//     Term 17 (AT2000-0250)/Term 18 (AT2000-5250)/FB Inputs/Value Channel 26 <-> Data Pointer/RawPositionValues[25]
//     Term 17 (AT2000-0250)/Term 18 (AT2000-5250)/FB Inputs/Value Channel 27 <-> Data Pointer/RawPositionValues[26]
//     Term 17 (AT2000-0250)/Term 18 (AT2000-5250)/FB Inputs/Value Channel 28 <-> Data Pointer/RawPositionValues[27]
//     Term 17 (AT2000-0250)/Term 18 (AT2000-5250)/FB Inputs/Value Channel 29 <-> Data Pointer/RawPositionValues[28]
//     Term 17 (AT2000-0250)/Term 18 (AT2000-5250)/FB Inputs/Value Channel 30 <-> Data Pointer/RawPositionValues[29]
//     Term 17 (AT2000-0250)/Term 18 (AT2000-5250)/FB Inputs/Value Channel 31 <-> Data Pointer/RawPositionValues[30]
//     Term 17 (AT2000-0250)/Term 18 (AT2000-5250)/FB Inputs/Value Channel 32 <-> Data Pointer/RawPositionValues[31]
//   NC-Task 1 SAF/Axes/Mover Axis 1 <-> TcCOM Objects/XTS ProcessingUnit 1/Mover 1
//     SoftDrive 1/Data Pointer/InputPointer1 <-> Inputs/SoftDriveInput
//     SoftDrive 1/Data Pointer/OutputPointer1 <-> Outputs/SoftDriveOutput
//   NC-Task 1 SAF/Axes/Mover Axis 2 <-> TcCOM Objects/XTS ProcessingUnit 1/Mover 2
//     SoftDrive 2/Data Pointer/InputPointer1 <-> Inputs/SoftDriveInput
//     SoftDrive 2/Data Pointer/OutputPointer1 <-> Outputs/SoftDriveOutput
//   NC-Task 1 SAF/Axes/Mover Axis 3 <-> TcCOM Objects/XTS ProcessingUnit 1/Mover 3
//     SoftDrive 3/Data Pointer/InputPointer1 <-> Inputs/SoftDriveInput
//     SoftDrive 3/Data Pointer/OutputPointer1 <-> Outputs/SoftDriveOutput
//   NC-Task 1 SAF/Axes/Mover Axis 4 <-> TcCOM Objects/XTS ProcessingUnit 1/Mover 4
//     SoftDrive 4/Data Pointer/InputPointer1 <-> Inputs/SoftDriveInput
//     SoftDrive 4/Data Pointer/OutputPointer1 <-> Outputs/SoftDriveOutput
//   NC-Task 1 SAF/Axes/Mover Axis 5 <-> TcCOM Objects/XTS ProcessingUnit 1/Mover 5
//     SoftDrive 5/Data Pointer/InputPointer1 <-> Inputs/SoftDriveInput
//     SoftDrive 5/Data Pointer/OutputPointer1 <-> Outputs/SoftDriveOutput
//   NC-Task 1 SAF/Axes/Mover Axis 6 <-> TcCOM Objects/XTS ProcessingUnit 1/Mover 6
//     SoftDrive 6/Data Pointer/InputPointer1 <-> Inputs/SoftDriveInput
//     SoftDrive 6/Data Pointer/OutputPointer1 <-> Outputs/SoftDriveOutput
//   XtsTransport/XtsTransport Instance <-> NC-Task 1 SAF/Axes/Conveyer
//     PlcTask Inputs/GVL_APPLICATION.MasterAxis.NcToPlc <-> Outputs/ToPlc
//     PlcTask Outputs/GVL_APPLICATION.MasterAxis.PlcToNc <-> Inputs/FromPlc
//   XtsTransport/XtsTransport Instance <-> NC-Task 1 SAF/Axes/Mover Axis 1
//     PlcTask Inputs/GVL_XTS.AxisRefMover[1].NcToPlc <-> Outputs/ToPlc
//     PlcTask Outputs/GVL_XTS.AxisRefMover[1].PlcToNc <-> Inputs/FromPlc
//   XtsTransport/XtsTransport Instance <-> NC-Task 1 SAF/Axes/Mover Axis 2
//     PlcTask Inputs/GVL_XTS.AxisRefMover[2].NcToPlc <-> Outputs/ToPlc
//     PlcTask Outputs/GVL_XTS.AxisRefMover[2].PlcToNc <-> Inputs/FromPlc
//   XtsTransport/XtsTransport Instance <-> NC-Task 1 SAF/Axes/Mover Axis 3
//     PlcTask Inputs/GVL_XTS.AxisRefMover[3].NcToPlc <-> Outputs/ToPlc
//     PlcTask Outputs/GVL_XTS.AxisRefMover[3].PlcToNc <-> Inputs/FromPlc
//   XtsTransport/XtsTransport Instance <-> NC-Task 1 SAF/Axes/Mover Axis 4
//     PlcTask Inputs/GVL_XTS.AxisRefMover[4].NcToPlc <-> Outputs/ToPlc
//     PlcTask Outputs/GVL_XTS.AxisRefMover[4].PlcToNc <-> Inputs/FromPlc
//   XtsTransport/XtsTransport Instance <-> NC-Task 1 SAF/Axes/Mover Axis 5
//     PlcTask Inputs/GVL_XTS.AxisRefMover[5].NcToPlc <-> Outputs/ToPlc
//     PlcTask Outputs/GVL_XTS.AxisRefMover[5].PlcToNc <-> Inputs/FromPlc
//   XtsTransport/XtsTransport Instance <-> NC-Task 1 SAF/Axes/Mover Axis 6
//     PlcTask Inputs/GVL_XTS.AxisRefMover[6].NcToPlc <-> Outputs/ToPlc
//     PlcTask Outputs/GVL_XTS.AxisRefMover[6].PlcToNc <-> Inputs/FromPlc
//   XtsTransport/XtsTransport Instance <-> NC-Task 1 SAF/Objects/Group1 (CA Group)
//     PlcTask Inputs/GVL_XTS.CaGroupRef.NcToPlc/CA <-> Group Outputs/ToPLC
//     PlcTask Outputs/GVL_XTS.CaGroupRef.PlcToNc/CA <-> Group Inputs/FromPLC

CONFIGURATION XtsTransport
    RESOURCE PLC ON TwinCAT3
        TASK PlcTask(INTERVAL := T#2ms, PRIORITY := 15);
        PROGRAM MAIN WITH PlcTask : MAIN;
        PROGRAM MAIN_APP WITH PlcTask : MAIN_APP;
    END_RESOURCE
END_CONFIGURATION

// ---- APPLICATION/_types/Instance/ST_INSTANCE_CTRL.TcDUT
{attribute 'pack_mode' := '2'}
TYPE ST_INSTANCE_CTRL :
STRUCT
  Cmd     : E_INSTANCE_CMD;
END_STRUCT
END_TYPE

// ---- APPLICATION/MAIN_APP.TcPOU
//---------------------------------------------------------------------------------------------------------------
//
//  HAUD 2024.10.02
//
//  - APPLICATION
//    - explicit simple example PRG for setting up GearInPosCa application
//      - works dirEctly on GVL_XTS namespace Ctrl/State structs
//      - no error handling, reset application from start
//
//  - Application controls:
//    - XtsTransport
//      - GVL_XTS.TransportCtrl
//      - GVL_XTS.TransportState
//
//    - Xts Movers
//      - GVL_XTS.MoverCtrl
//      - GVL_XTS.MoverState
//      - GVL_XTS.MoverInfo
//      - GVL_XTS.MoveData
//      - GVL_XTS.GearData
//
//  - Application
//    - GearInPosCa example
//      - gear in to conveyer belt 
//
//---------------------------------------------------------------------------------------------------------------
// This SOFTWARE is provided as an Exemple by THE PROVIDER "as is" and "with all faults." THE PROVIDER makes no 
// representations or warranties of any kind concerning the safety, suitability, lack of viruses, inaccuracies, 
// typographical errors, or other harmful components of this SOFTWARE. There are inherent dangers in the use of 
// any software, and you are solely responsible for determining whether this SOFTWARE is compatible with your 
// equipment and other software installed on your equipment. You are also solely responsible for the protection 
// of your equipment and backup of your data, and THE PROVIDER will not be liable for any damages you may suffer 
// in connection with using, modifying, or distributing this SOFTWARE.
//---------------------------------------------------------------------------------------------------------------
PROGRAM MAIN_APP
VAR
  eInit         : E_PROGRESS;
  bStart        : BOOL;   // XtsTransport is initialized, CAGroup is built, All movers are enabled, XtsStations are cleared, XtsTransport base position for all movers is commanded, XtsStations are handshaked with timer
  bReset        : BOOL;   // All Xts Stations are cleared, requires new start

  nState        : UINT;   // state var for application
END_VAR



//-----------------------------------------------------------------------------
// wait for initialization to be complete before work may start
//-----------------------------------------------------------------------------
IF NOT (MAIN_XTS.eInit = E_PROGRESS.PROGRESS_DONE)
THEN
  eInit                               := E_PROGRESS.PROGRESS_INIT;
  bReset                              := FALSE;
  bStart                              := FALSE;
  nState                              := 0;
  RETURN;
END_IF
//-----------------------------------------------------------------------------
// fetch reset anytime
//-----------------------------------------------------------------------------
IF bReset
THEN
  bReset                              := FALSE;
  bStart                              := FALSE;
  nState                              := 9000;  // states for clearing XtsTransport
END_IF


CASE nState 
OF
  0:                                  // first PLC cycle
    nState                            := 1;

  1:
    // do other init stuff here
    eInit                             := E_PROGRESS.PROGRESS_DONE;
    nState                            := 10;

  10:                                 // starts from here
    IF bStart
    THEN
      nState                          := 100; // let's go
    END_IF
    
  100:                                // clear interface
    GVL_XTS.XtsTransportCtrl.Cmd      := E_XTS_TRANSPORT_CTRL.CMD_NULL;
    nState                            := 110;

  110:                                // check initialization of XtsTransport, wait for either MoverDetection being valid or OperationMode.Simulation
    IF (GVL_XTS.XtsTransportState.XpuInfo.IdDetectionValid) OR
       (GVL_XTS.XtsTransportState.XpuInfo.OperationMode = OperationMode.Simulation)
    THEN
      // now XtsTransport is initialized, cyclic plausibility checks on Xpu are active
      nState                          := 120;
    END_IF

  120:                                // clear group for defined start situation
    GVL_XTS.XtsTransportCtrl.Cmd      := E_XTS_TRANSPORT_CTRL.CMD_GROUP_CLEAR;

    IF (GVL_XTS.XtsTransportState.State = E_XTS_TRANSPORT_STATE.TRANSPORT_GROUP_CLEAR + E_PROGRESS.PROGRESS_DONE)
    THEN
      // CA Group is now in defined error free state
      nState                          := 130;
    END_IF

  130:                                // build Collision Avoidance group with all movers
    GVL_XTS.XtsTransportCtrl.Cmd      := E_XTS_TRANSPORT_CTRL.CMD_GROUP_BUILD;

    IF (GVL_XTS.XtsTransportState.State = E_XTS_TRANSPORT_STATE.TRANSPORT_GROUP_BUILD + E_PROGRESS.PROGRESS_DONE)
    THEN
      // CA Group contains all movers now
      // GVL_XTS.XtsTransportState.GroupInfo.AxisCount = MAX_MOVER
      nState                          := 140;
      GEAR_IN_POS_CA.bEnable          := FALSE;
      GEAR_IN_POS_CA.bReset           := FALSE;
    END_IF

  140:                                // enable CA Group
    GVL_XTS.XtsTransportCtrl.Cmd      := E_XTS_TRANSPORT_CTRL.CMD_GROUP_ENABLE;

    IF (GVL_XTS.XtsTransportState.State = E_XTS_TRANSPORT_STATE.TRANSPORT_GROUP_ENABLE + E_PROGRESS.PROGRESS_DONE)
    THEN
      // GVL_XTS.XtsTransportState.GroupInfo.CaGroupState = mcGroupStateNotReady
      nState                          := 150;
      GEAR_IN_POS_CA.bReset           := TRUE;
    END_IF

  150:                                // enable all movers
    GVL_XTS.XtsTransportCtrl.Cmd      := E_XTS_TRANSPORT_CTRL.CMD_MOVER_ENABLE;

    IF (GVL_XTS.XtsTransportState.State = E_XTS_TRANSPORT_STATE.TRANSPORT_MOVER_ENABLE + E_PROGRESS.PROGRESS_DONE)
    THEN
      // GVL_XTS.XtsTransportState.GroupInfo.CaGroupState = mcGroupStateStandby
      nState                          := 160;
      GEAR_IN_POS_CA.bReset           := FALSE;
    END_IF

  160:                                // command all movers to startup position
    GVL_XTS.XtsTransportCtrl.Cmd      := E_XTS_TRANSPORT_CTRL.CMD_TRANSPORT_START;

    IF (GVL_XTS.XtsTransportState.State = E_XTS_TRANSPORT_STATE.TRANSPORT_START + E_PROGRESS.PROGRESS_DONE)
    THEN
      // all movers are now waiting at GVL_XTS.StationStart.rPosWait
      nState                          := 1000; // go to wait state, activate GearInPos program
      // enable gear in pos sequence now the movers are ready
      GEAR_IN_POS_CA.bEnable          := TRUE;
    END_IF


  9000:
    // reset sequence trigger starts here
    GEAR_IN_POS_CA.bEnable            := FALSE;
    GVL_XTS.XtsTransportCtrl.Cmd      := E_XTS_TRANSPORT_CTRL.CMD_NULL;
    nState                            := 9005;

    GVL_APPLICATION.MasterHalt(
                        Axis          := GVL_APPLICATION.MasterAxis, 
                        Execute       := FALSE, 
                        Deceleration  :=  12500.0, 
                        Jerk          := 100000.0, 
                        BufferMode    := Tc2_MC2.MC_Aborting, 
                        Options:= , 
                        Done=> , 
                        Busy=> , 
                        Active=> , 
                        CommandAborted=> , 
                        Error=> , 
                        ErrorID=> );

  9005:
    GVL_APPLICATION.MasterHalt(
                        Axis          := GVL_APPLICATION.MasterAxis, 
                        Execute       := TRUE);

    IF (GVL_APPLICATION.MasterAxis.Status.NotMoving)
    THEN
      nState                          := 9010;

      GVL_APPLICATION.MasterHalt(
                          Axis        := GVL_APPLICATION.MasterAxis, 
                          Execute     := FALSE);

      GVL_APPLICATION.MasterPower(
                  Axis                := GVL_APPLICATION.MasterAxis, 
                  Enable              := FALSE);
    END_IF

  9010:                               // halt all movers and clear group
    GVL_XTS.XtsTransportCtrl.Cmd      := E_XTS_TRANSPORT_CTRL.CMD_GROUP_CLEAR;

    IF (GVL_XTS.XtsTransportState.State = E_XTS_TRANSPORT_STATE.TRANSPORT_GROUP_CLEAR + E_PROGRESS.PROGRESS_DONE)
    THEN
      // CA group cleared and mover in standstill
      nState                          := 9100;
    END_IF

  9100:                               // switch off movers
    GVL_XTS.XtsTransportCtrl.Cmd      := E_XTS_TRANSPORT_CTRL.CMD_MOVER_DISABLE;

    IF (GVL_XTS.XtsTransportState.State = E_XTS_TRANSPORT_STATE.TRANSPORT_MOVER_DISABLE + E_PROGRESS.PROGRESS_ERROR)
    THEN
      nState                          := 9010;
    ELSIF (GVL_XTS.XtsTransportState.State = E_XTS_TRANSPORT_STATE.TRANSPORT_MOVER_DISABLE + E_PROGRESS.PROGRESS_DONE)
    THEN
      nState                          := 10;
    END_IF

END_CASE

GVL_APPLICATION.MasterAxis(); // update master axis

GEAR_IN_POS_CA();             // gear in pos sequence

END_PROGRAM

// ---- APPLICATION/GEAR_IN_POS_CA.TcPOU
//---------------------------------------------------------------------------------------------------------------
//
//  HAUD 2024.10.02
//
//  - simple program for GearInPosCa of mover and conveyer belt (MasterAxis)
//    - mover is geared in
//    - sync distance is checked
//    - mover is sent to target position
//---------------------------------------------------------------------------------------------------------------
PROGRAM GEAR_IN_POS_CA
VAR_INPUT
  bReset                : BOOL;
  bEnable               : BOOL;
END_VAR
VAR_OUTPUT
  bError                : BOOL;
END_VAR
VAR
  nErrorId              : UDINT;

  // this example checks the sync distance of the conveyer
  rDiffPositionConveyer, 
  rStartPositionConveyer,
  rTargetPositionMover  : LREAL;

  rSyncDistance         : LREAL;
  rSyncDistanceConveyer : LREAL := 225.0;

  nState                : UINT;
  nMover                : UINT;
  rtrigReset            : Tc2_Standard.R_TRIG;
END_VAR

rtrigReset(CLK:= bReset);
IF rtrigReset.Q
THEN
  nState                       := 0;
  FOR nMover := 1 TO MAX_MOVER
  DO
    GVL_XTS.MoverCtrl[nMover].Cmd      := E_MOVER_CTRL.MOVER_NULL;
  END_FOR
END_IF





CASE nState OF
  0:
    IF bEnable AND NOT bReset
    THEN
      bError                        := FALSE;
      nErrorId                      := 0;
      nMover                        := 1;
      nState                        := 10;
    END_IF

  10:
    nState                          := 11;
    GVL_APPLICATION.MasterReset(
                      Axis          := GVL_APPLICATION.MasterAxis, 
                      Execute       := FALSE, 
                      Done=> , 
                      Busy=> , 
                      Error=> , 
                      ErrorID=> );

  11:
    GVL_APPLICATION.MasterReset(
                      Axis          := GVL_APPLICATION.MasterAxis, 
                      Execute       := TRUE);

    IF (GVL_APPLICATION.MasterReset.Done)
    THEN
      nState                        := 12;
    END_IF

  12:
    nState                          := 13;
    GVL_APPLICATION.MasterReset(
                      Axis          := GVL_APPLICATION.MasterAxis, 
                      Execute       := FALSE);

  13:
    GVL_APPLICATION.MasterPower(
                Axis                := GVL_APPLICATION.MasterAxis, 
                Enable              := TRUE, 
                Enable_Positive     := TRUE, 
                Enable_Negative     := TRUE, 
                Override            := GVL_APPLICATION.MoveData.rOverride, 
                BufferMode:= , 
                Options:= , 
                Status=> , 
                Busy=> , 
                Error=> , 
                ErrorID=> );

    IF NOT (GVL_APPLICATION.MasterPower.Error)
    THEN
      IF (GVL_APPLICATION.MasterAxis.Status.ControlLoopClosed)
      THEN
        nState                      := 14;
      END_IF
    ELSE
      nState                        := 9000;
      nErrorId                      := GVL_APPLICATION.MasterPower.ErrorID;
    END_IF

  14:
    nState                          := 15;

    // READ THIS:
    // https://infosys.beckhoff.com/english.php?content=../content/1033/tf5410_tc3_collision_avoidance/1534969995.html&id=

    GVL_APPLICATION.MoveData.rVelo  :=  1000.0;   // dynamics for gearing procedure
    GVL_APPLICATION.MoveData.rAcc   := 12500.0;   // dynamics for gearing procedure
    GVL_APPLICATION.MoveData.rGap   :=   100.0;   // gap which has to be maintained during operations

    GVL_APPLICATION.GearData.rDeltaToMasterPos      :=  125.0;  // distance to GearIn position of master
    GVL_APPLICATION.GearData.rMasterStartDistance   :=    0.0;  // distance master has to move until gearing is started
    GVL_APPLICATION.GearData.rModuloSyncPosSlave    :=   75.0;  // Modulo Position of mover where master and mover have to be in sync
    GVL_APPLICATION.GearData.rGearNumerator         :=    1.0;  // Gearing factor

    GVL_APPLICATION.MasterMoveVelo(
                  Axis              := GVL_APPLICATION.MasterAxis, 
                  Execute           := FALSE, 
                  Velocity          :=    500.0, 
                  Acceleration      :=  12500.0, 
                  Deceleration      :=  12500.0, 
                  Jerk              := 100000.0, 
                  Direction         := Tc2_MC2.MC_Direction.MC_Positive_Direction, 
                  BufferMode        := Tc2_MC2.MC_Aborting, 
                  Options:= , 
                  InVelocity=> , 
                  Busy=> , 
                  Active=> , 
                  CommandAborted=> , 
                  Error=> , 
                  ErrorID=> );

  15:
    GVL_APPLICATION.MasterMoveVelo(
                  Axis              := GVL_APPLICATION.MasterAxis, 
                  Execute           := TRUE);

    IF (GVL_APPLICATION.MasterMoveVelo.Error)
    THEN
      nState                        := 9000;
      nErrorId                      := GVL_APPLICATION.MasterMoveVelo.ErrorID;

    ELSIF (GVL_APPLICATION.MasterMoveVelo.InVelocity)
    THEN
      nState                        := 1000;
    END_IF


  1000:
    IF bEnable
    THEN
      nState                        := 1010;
      // see method fb_Mover.GearInPosCa for how the MC_GearInPosCa is connected
      // GVL_XTS.MoverCtrl is triggering fb_MoverCtrl(fb_Mover) instance
      GVL_XTS.Mover[nMover].Master  ref= GVL_APPLICATION.MasterAxis;
      GVL_XTS.MoveData [nMover]     := GVL_APPLICATION.MoveData;  // feed dynamic constraints into datafield of mover
      GVL_XTS.GearData [nMover]     := GVL_APPLICATION.GearData;  // feed gearing constraints into datafield of mover

      GVL_XTS.MoverCtrl[nMover].Cmd := E_MOVER_CTRL.MOVER_GEAR_IN_POS_CA; // start gearing procedure 
    END_IF

  1010:
    IF (GVL_XTS.MoverState[nMover].State = E_MOVER_STATE.MOVER_GEAR_IN_POS_CA + E_PROGRESS.PROGRESS_ERROR)
    THEN
      nErrorId                      := GVL_XTS.MoverInfo[nMover].nErrorId;
      nState                        := 9000;

    ELSIF (GVL_XTS.MoverState[nMover].State = E_MOVER_STATE.MOVER_GEAR_IN_POS_CA + E_PROGRESS.PROGRESS_DONE)
    THEN
      // sync movement is reached, now check for SyncDistance and then send mover away
      nState                        := 1020;
      rDiffPositionConveyer         := GVL_APPLICATION.MasterAxis.NcToPlc.ActPos - rStartPositionConveyer;
      rStartPositionConveyer        := GVL_APPLICATION.MasterAxis.NcToPlc.ActPos;
      rTargetPositionMover          := GVL_XTS.MoverItf [nMover].RailLength + GVL_XTS.StationStart.rPosWait; // this example sends movers one RailLength forward to startup position 
    END_IF

  1020:
    rSyncDistance                   := GVL_APPLICATION.MasterAxis.NcToPlc.ActPos - rStartPositionConveyer;
    IF (rSyncDistance > rSyncDistanceConveyer)
    THEN
      // sync distance is reached, now send mover away
      nState                              := 1030;
      GVL_XTS.MoveData [nMover].rPos      := rTargetPositionMover;
      GVL_XTS.MoveData [nMover].rGap      := GVL_XTS.StationStart.rGap;
      GVL_XTS.MoveData [nMover].rDistance := -5.0; // mover has to move more than this distance, then E_MOVER_CTRL.MOVER_SEND_TO_POS_CA is done

      GVL_XTS.MoverCtrl[nMover].Cmd := E_MOVER_CTRL.MOVER_SEND_TO_POS_CA;
    END_IF

  1030:
    IF (GVL_XTS.MoverState[nMover].State = E_MOVER_STATE.MOVER_SEND_TO_POS_CA + E_PROGRESS.PROGRESS_ERROR)
    THEN
      nErrorId                      := GVL_XTS.MoverInfo[nMover].nErrorId;
      nState                        := 9000;

    ELSIF (GVL_XTS.MoverState[nMover].State = E_MOVER_STATE.MOVER_SEND_TO_POS_CA + E_PROGRESS.PROGRESS_DONE)
    THEN
      nState                        := 1040;
    END_IF

  1040:
    nState                          := 1000;
    IF (nMover > MAX_MOVER-1)
    THEN
      nMover                        := 1;
    ELSE
      nMover                        := nMover + 1;
    END_IF

  9000:
    bError                          := TRUE;
END_CASE

END_PROGRAM

// ---- APPLICATION/_types/Collector/fb_ProcessCollector.TcPOU
//---------------------------------------------------------------------------------------------------------------
//
//  HAUD 2024.10.13
//
//
//  fb_ProcessCollector
//  - wraps range of XtsStations for parallel processes
//  - sets process states for extern control (Ctrl/State)
//  - conveys command onto XtsStations
//  
//
//---------------------------------------------------------------------------------------------------------------//
// This SOFTWARE is provided as an Example by THE PROVIDER "as is" and "with all faults." THE PROVIDER makes no  //
// representations or warranties of any kind concerning the safety, suitability, lack of viruses, inaccuracies,  //
// typographical errors, or other harmful components of this SOFTWARE. There are inherent dangers in the use of  //
// any software, and you are solely responsible for determining whether this SOFTWARE is compatible with your    //
// equipment and other software installed on your equipment. You are also solely responsible for the protection  //
// of your equipment and backup of your data, and THE PROVIDER will not be liable for any damages you may suffer //
// in connection with using, modifying, or distributing this SOFTWARE.                                           //
//---------------------------------------------------------------------------------------------------------------//
FUNCTION_BLOCK fb_ProcessCollector EXTENDS fb_StationCollector IMPLEMENTS I_ProcessCollector
VAR

  _stControl      : REFERENCE TO ST_PROCESS_CTRL;  // ctrl via property
  _stState        : REFERENCE TO ST_PROCESS_STATE; // state via property

  _eCmd,                              // command for controlling the XtsStations
  _eCmdOld        : E_PROCESS_CTRL;   // logging of command on change
  _eStateProgress : E_PROGRESS;       // progress sub state for process
  _eResult        : E_PROGRESS;       // progress result for methods

  // ctrl words for XtsStations
  {attribute 'displaymode':='bin'}
  _wActivateStation     : T_PROCESS;  // bits enable XtsStations in this process, that's what drives me

  // ctrl data for used target XtsStations in target process
  {attribute 'displaymode':='bin'}
  _wTargetMask          : ARRAY[1..SIZEOF(T_PROCESS)*8] OF BYTE;    // mask for multiple PosStop in target
  _rTargetOffset        : ARRAY[1..SIZEOF(T_PROCESS)*8] OF LREAL;   // dyn offset for mulriple PosStop in target

  _nTargetIndex         : ARRAY[1..SIZEOF(T_PROCESS)*8] OF USINT;   // index of XtsStation in target process

  // debug / scope vars for ctrl on XtsStation
  // one bit: one XtsStation
  {attribute 'displaymode':='bin'}
  _wCtrlEnable          : T_PROCESS;
  {attribute 'displaymode':='bin'}
  _wCtrlEnter           : T_PROCESS;
  {attribute 'displaymode':='bin'}
  _wCtrlSend            : T_PROCESS;
  {attribute 'displaymode':='bin'}
  _wCtrlStart           : T_PROCESS;
  {attribute 'displaymode':='bin'}
  _wCtrlDone            : T_PROCESS;
  {attribute 'displaymode':='bin'}
  _wCtrlNest            : T_PROCESS;
  {attribute 'displaymode':='bin'}
  _wCtrlOut             : T_PROCESS;
END_VAR

PROPERTY ActivateStation : DWORD // bit mask for enabling XtsStations in Process
GET
ActivateStation := _wActivateStation;
END_GET
END_PROPERTY

METHOD PRIVATE Controls // called in Cycle(), conveys single process command to range of XtsStations
VAR_INPUT
  Cmd       : E_PROCESS_CTRL;
END_VAR
VAR
  _idx      : UINT;
END_VAR

FOR _idx := _nStationLast TO _nStationFirst BY(-1)
DO
  CASE _stStationState[_idx].State
  OF
    //-------------------------------------------------------------------------
    E_STATION_STATE.STATION_DISABLE:
      CASE Cmd
      OF
        E_PROCESS_CTRL.PROCESS_ENABLE:    // switch on
          IF (_wActivateStation > 0)      // must be at least one XtsStation to switch on
          THEN
            // check who to switch on
            IF (BitGet(_wActivateStation, (_idx - _nStationFirst)))
            THEN
              _stStationCtrl[_idx].Cmd     := E_STATION_CTRL.STATION_ENABLE;

              // clear XtsStation ctrl interface, must be written before movers are sent out 
              // see below (STATION_MOVER_OUT) from where those values have to come
              _stStationCtrl[_idx].nMask          := 0;
              _stStationCtrl[_idx].rOffset        := 0;
              _stStationCtrl[_idx].nTargetStation := 0;

              _wCtrlEnable                := BitSet(_wCtrlEnable, (_idx - _nStationFirst)); 

              _wCtrlEnter                 := BitDel(_wCtrlEnter,  (_idx - _nStationFirst));
              _wCtrlSend                  := BitDel(_wCtrlSend,   (_idx - _nStationFirst));
              _wCtrlStart                 := BitDel(_wCtrlStart,  (_idx - _nStationFirst));
              _wCtrlDone                  := BitDel(_wCtrlDone,   (_idx - _nStationFirst));
              _wCtrlNest                  := BitDel(_wCtrlNest,   (_idx - _nStationFirst));
              _wCtrlOut                   := BitDel(_wCtrlOut,    (_idx - _nStationFirst));
            END_IF
          END_IF
      END_CASE

    //-------------------------------------------------------------------------
    E_STATION_STATE.STATION_ENABLE,
    E_STATION_STATE.STATION_DETECT_MOVER:
      CASE Cmd
      OF
        E_PROCESS_CTRL.PROCESS_DISABLE:
          _wCtrlEnable                    := BitDel(_wCtrlEnable, (_idx - _nStationFirst));
          _stStationCtrl[_idx].Cmd         := E_STATION_CTRL.STATION_DISABLE;

        E_PROCESS_CTRL.PROCESS_ENABLE:
          _wCtrlEnable                    := BitSet(_wCtrlEnable, (_idx - _nStationFirst));
          _stStationCtrl[_idx].Cmd         := E_STATION_CTRL.STATION_ENABLE;
      END_CASE

    //-------------------------------------------------------------------------
    E_STATION_STATE.STATION_MOVER_ENTER:
      CASE Cmd
      OF
        E_PROCESS_CTRL.PROCESS_DISABLE:
          _wCtrlEnable                    := BitDel(_wCtrlEnable, (_idx - _nStationFirst));
          _stStationCtrl[_idx].Cmd         := E_STATION_CTRL.STATION_DISABLE;

        E_PROCESS_CTRL.PROCESS_ENABLE:
          _wCtrlEnable                    := BitSet(_wCtrlEnable, (_idx - _nStationFirst));
          _stStationCtrl[_idx].Cmd         := E_STATION_CTRL.STATION_ENABLE;

        E_PROCESS_CTRL.PROCESS_STATIONS_ENTER:
          _wCtrlEnter                     := BitSet(_wCtrlEnter, (_idx - _nStationFirst));
          _stStationCtrl[_idx].Cmd         := E_STATION_CTRL.STATION_MOVER_ENTER;

        E_PROCESS_CTRL.PROCESS_STATIONS_SEND:
          _wCtrlSend                      := BitSet(_wCtrlSend, (_idx - _nStationFirst));
          _stStationCtrl[_idx].Cmd         := E_STATION_CTRL.STATION_MOVER_SEND;
      END_CASE

    //-------------------------------------------------------------------------
    E_STATION_STATE.STATION_PROCESS_START:
      CASE Cmd
      OF
        E_PROCESS_CTRL.PROCESS_START:
          _wCtrlStart                     := BitSet(_wCtrlStart,  (_idx - _nStationFirst));
          _stStationCtrl[_idx].Cmd         := E_STATION_CTRL.STATION_PROCESS_START;

        E_PROCESS_CTRL.PROCESS_DONE:
          _wCtrlDone                      := BitSet(_wCtrlDone,   (_idx - _nStationFirst));
          _stStationCtrl[_idx].Cmd         := E_STATION_CTRL.STATION_PROCESS_DONE;
      END_CASE

    //-------------------------------------------------------------------------
    E_STATION_STATE.STATION_PROCESS_DONE:
      _stStationCtrl[_idx].nMask            :=          _wTargetMask  [1+_idx - _nStationFirst];
      _stStationCtrl[_idx].rOffset          := TO_REAL( _rTargetOffset[1+_idx - _nStationFirst]);
      _stStationCtrl[_idx].nTargetStation   :=          _nTargetIndex [1+_idx - _nStationFirst];

      CASE Cmd
      OF
        E_PROCESS_CTRL.PROCESS_DONE:
          _wCtrlDone                      := BitSet(_wCtrlDone,   (_idx - _nStationFirst));
          _stStationCtrl[_idx].Cmd         := E_STATION_CTRL.STATION_PROCESS_DONE;

        E_PROCESS_CTRL.PROCESS_STATIONS_OUTFEED:
          _wCtrlDone                      := BitSet(_wCtrlDone,   (_idx - _nStationFirst));
          _stStationCtrl[_idx].Cmd         := E_STATION_CTRL.STATION_MOVER_OUT;
      END_CASE

    //-------------------------------------------------------------------------
    E_STATION_STATE.STATION_CHECK_NEST:
      CASE Cmd
      OF
        E_PROCESS_CTRL.PROCESS_STATIONS_ENTER:
          _wCtrlStart                     := BitDel(_wCtrlStart,  (_idx - _nStationFirst));
          _wCtrlNest                      := BitSet(_wCtrlNest,   (_idx - _nStationFirst));
          _stStationCtrl[_idx].Cmd         := E_STATION_CTRL.STATION_MOVER_ENTER;
      END_CASE

    //-------------------------------------------------------------------------
    E_STATION_STATE.STATION_MOVER_OUT:
      _stStationCtrl[_idx].nMask            :=          _wTargetMask  [1+_idx - _nStationFirst];
      _stStationCtrl[_idx].rOffset          := TO_REAL( _rTargetOffset[1+_idx - _nStationFirst]);
      _stStationCtrl[_idx].nTargetStation   :=          _nTargetIndex [1+_idx - _nStationFirst];

      CASE Cmd
      OF
        E_PROCESS_CTRL.PROCESS_STATIONS_OUTFEED:
          _wCtrlOut                       := BitSet(_wCtrlOut,    (_idx - _nStationFirst));
          _stStationCtrl[_idx].Cmd         := E_STATION_CTRL.STATION_MOVER_OUT;
      END_CASE

    //-------------------------------------------------------------------------
    E_STATION_STATE.STATION_MOVER_GONE:
      _wCtrlEnable                        := BitDel(_wCtrlEnable, (_idx - _nStationFirst));
      _wCtrlEnter                         := BitDel(_wCtrlEnter,  (_idx - _nStationFirst));
      _wCtrlSend                          := BitDel(_wCtrlSend,   (_idx - _nStationFirst));
      _wCtrlStart                         := BitDel(_wCtrlStart,  (_idx - _nStationFirst));
      _wCtrlDone                          := BitDel(_wCtrlDone,   (_idx - _nStationFirst));
      _wCtrlNest                          := BitDel(_wCtrlNest,   (_idx - _nStationFirst));

      _stStationCtrl[_idx].Cmd             := E_STATION_CTRL.STATION_MOVER_GONE;

  END_CASE
END_FOR
END_METHOD

METHOD PUBLIC Cycle // cyclic call for checking XtsStation state masks and command input from process
//-------------------------------------------------------------------------------------------------
//-------------------------------------------------------------------------------------------------
//  HAUD 2024 10 21
//  cyclic call required
//
//-------------------------------------------------------------------------------------------------
//-------------------------------------------------------------------------------------------------
// reference checks
//-------------------------------------------------------------------------------------------------
IF NOT __ISVALIDREF(_stControl)
THEN
  _eCheck                           := E_PROCESS_CHECK.REFERENCE_CTRL_INVALID;
  RETURN;
END_IF

IF NOT __ISVALIDREF(_stState)
THEN
  _eCheck                           := E_PROCESS_CHECK.REFERENCE_STATE_INVALID;
  RETURN;
END_IF
//-------------------------------------------------------------------------------------------------
//-------------------------------------------------------------------------------------------------
// plausibility checks
//-------------------------------------------------------------------------------------------------
IF NOT Check()
THEN
  // you shall not pass!!
  RETURN;
END_IF
//-------------------------------------------------------------------------------------------------
//-------------------------------------------------------------------------------------------------
// Message device identification
//-------------------------------------------------------------------------------------------------
_stMsg.eDevice                      := e_Device.Process + TO_UINT(_nProcessId);
//-------------------------------------------------------------------------------------------------
//-------------------------------------------------------------------------------------------------
// XtsStation states:
//  - fb_ProcessCollector extends fb_StationCollector: 
//    --> cyclic call of States() for getting station masks
//
//  - sets bit for every XtsStation
//-------------------------------------------------------------------------------------------------
//
States();                           // not just mental, literal
//-------------------------------------------------------------------------------------------------
//-------------------------------------------------------------------------------------------------
// process states
//-------------------------------------------------------------------------------------------------
CASE _stState.State
OF
  //-----------------------------------------------------------------------------------------------
  E_PROCESS_STATE.PROCESS_DISABLE:  // default wait state
    //-------------------------------------------------------------------------
    CASE _eStateProgress            // check if all my XtsStations are disabled
    OF
      E_PROGRESS.PROGRESS_INIT:
        IF (_wStateDisable = EXPT(2,_nStationCount)-1)                  // all stations in process range must be disabled at this point
        THEN
          // on a sunny afternoon, nothing to do, just sit and wait
          _eStateProgress           := E_PROGRESS.PROGRESS_BUSY;

          IF (_MessageLevel > E_MessageType.eMessageInfo)
          THEN
            _stMsg.eType            := E_MessageType.eMessageVerbose;
            _stMsg.eSubdevice       := e_Subdevice.Process_ProcessCollector_Cycle;
            _stMsg.iErrorNumber     := _wStateDisable;
            _stMsg.sText            := concat('_wStateDisable: ', BitsToString(_wStateDisable));
            _stMsg.sText            := concat(_stMsg.sText, ': ');
            _stMsg.sText            := concat(_stMsg.sText, TO_STRING(_eStateProgress));
            f_MessageSet(_stMsg);
          END_IF
        END_IF
    END_CASE
    //-------------------------------------------------------------------------
    CASE _eStateProgress            // check for process enable signal
    OF
      E_PROGRESS.PROGRESS_BUSY:
      CASE _stControl.Cmd                                               // check process command
      OF
        E_PROCESS_CTRL.PROCESS_ENABLE:                                  // only one thing to say here..
          _eCmd                     := _stControl.Cmd;                  // copy command from interface to local switch
          // you do what I say, when I say it
          _wActivateStation         := _stControl.ActivateStation;      // on enabling of process, copy my active stations from interface

          LogControl(_eCmd);

          _eStateProgress           := E_PROGRESS.PROGRESS_INIT;        // switch back sub state
          _stState.State            := E_PROCESS_STATE.PROCESS_ENABLE;  // switch to enable

          IF (_MessageLevel > E_MessageType.eMessageError)
          THEN
            _stMsg.eType            := E_MessageType.eMessageInfo;
            _stMsg.eSubdevice       := e_Subdevice.Process_ProcessCollector_Cycle;
            _stMsg.iErrorNumber     := _nProcessId;
            _stMsg.sText            := concat(TO_STRING(_stState.State), ': ');
            _stMsg.sText            := concat(_stMsg.sText, TO_STRING(_eStateProgress));
            f_MessageSet(_stMsg);
          END_IF
      END_CASE
    END_CASE
END_CASE
//-------------------------------------------------------------------------------------------------
//-------------------------------------------------------------------------------------------------
CASE _stState.State
OF
  //-----------------------------------------------------------------------------------------------
  E_PROCESS_STATE.PROCESS_ENABLE:   // wait here for process command "allow infeed"
    //-------------------------------------------------------------------------
    CASE _eStateProgress
    OF
      E_PROGRESS.PROGRESS_INIT:
        IF (_wStateEnable = _wActivateStation)                          // all active stations must be enabled
        THEN
          // we are truly equal, yet not the same
          _eStateProgress           := E_PROGRESS.PROGRESS_BUSY;

          IF (_MessageLevel > E_MessageType.eMessageInfo)
          THEN
            _stMsg.eType            := E_MessageType.eMessageVerbose;
            _stMsg.eSubdevice       := e_Subdevice.Process_ProcessCollector_Cycle;
            _stMsg.iErrorNumber     := _wStateEnable;
            _stMsg.sText            := concat('_wStateEnable: ', BitsToString(_wStateEnable));
            _stMsg.sText            := concat(_stMsg.sText, ': ');
            _stMsg.sText            := concat(_stMsg.sText, TO_STRING(_eStateProgress));
            f_MessageSet(_stMsg);
          END_IF
        END_IF
    END_CASE
    //-------------------------------------------------------------------------
    CASE _eStateProgress
    OF
      E_PROGRESS.PROGRESS_BUSY:
      // check command for further instructions
      CASE _stControl.Cmd
      OF
        E_PROCESS_CTRL.PROCESS_DISABLE:                                 // command decided to switch OFF  
          _eCmd                     := _stControl.Cmd;                  // copy command from interface

          LogControl(_eCmd);

          _eStateProgress           := E_PROGRESS.PROGRESS_INIT;        // switch back sub state
          _stState.State            := E_PROCESS_STATE.PROCESS_DISABLE;

          IF (_MessageLevel > E_MessageType.eMessageInfo)
          THEN
            _stMsg.eType            := E_MessageType.eMessageVerbose;
            _stMsg.eSubdevice       := e_Subdevice.Process_ProcessCollector_Cycle;
            _stMsg.iErrorNumber     := _nProcessId;
            _stMsg.sText            := concat(TO_STRING(_stState.State), ': ');
            _stMsg.sText            := concat(_stMsg.sText, TO_STRING(_eStateProgress));
            f_MessageSet(_stMsg);
          END_IF


        E_PROCESS_CTRL.PROCESS_STATIONS_INFEED,
        E_PROCESS_CTRL.PROCESS_STATIONS_ENTER,
        E_PROCESS_CTRL.PROCESS_STATIONS_SEND:                           // command decided to allow checking the infeed into process
          _eStateProgress           := E_PROGRESS.PROGRESS_INIT;        // switch back sub state
          _stState.State            := E_PROCESS_STATE.PROCESS_STATIONS_INFEED;

          IF (_MessageLevel > E_MessageType.eMessageWarning)
          THEN
            _stMsg.eType            := E_MessageType.eMessageInfo;
            _stMsg.eSubdevice       := e_Subdevice.Process_ProcessCollector_Cycle;
            _stMsg.iErrorNumber     := _nProcessId;
            _stMsg.sText            := concat(TO_STRING(_stState.State), ': ');
            _stMsg.sText            := concat(_stMsg.sText, TO_STRING(_eStateProgress));
            f_MessageSet(_stMsg);
          END_IF
      END_CASE
    END_CASE
END_CASE
//-------------------------------------------------------------------------------------------------
//-------------------------------------------------------------------------------------------------
CASE _stState.State
OF
  //-----------------------------------------------------------------------------------------------
  E_PROCESS_STATE.PROCESS_STATIONS_INFEED:  // wait state for checking infeed command
    //-------------------------------------------------------------------------
    CASE _eStateProgress
    OF
      E_PROGRESS.PROGRESS_INIT:
        IF (_wStateEnter = _wActivateStation)                           // all active XtsStations must have mover waiting
        THEN
          // mover IDs are known by now --> Check _nMoverIdQueue for your plausibility checks
          // master master, there's the thing I've been after
          _eStateProgress           := E_PROGRESS.PROGRESS_BUSY;

          IF (_MessageLevel > E_MessageType.eMessageInfo)
          THEN
            _stMsg.eType            := E_MessageType.eMessageVerbose;
            _stMsg.eSubdevice       := e_Subdevice.Process_ProcessCollector_Cycle;
            _stMsg.iErrorNumber     := _wStateEnter;
            _stMsg.sText            := concat('_wStateEnter: ', BitsToString(_wStateEnter));
            _stMsg.sText            := concat(_stMsg.sText, ': ');
            _stMsg.sText            := concat(_stMsg.sText, TO_STRING(_eStateProgress));
            f_MessageSet(_stMsg);
          END_IF
        END_IF
    END_CASE
    //-------------------------------------------------------------------------
    CASE _eStateProgress
    OF
      E_PROGRESS.PROGRESS_BUSY:
      CASE _stControl.Cmd                                               // check command from interface
      OF
        E_PROCESS_CTRL.PROCESS_STATIONS_ENTER:
          _eCmd                     := _stControl.Cmd;                  // copy command to start infeed of movers

          LogControl(_eCmd);

          _eStateProgress           := E_PROGRESS.PROGRESS_INIT;        // switch back sub state
          _stState.State            := E_PROCESS_STATE.PROCESS_START;

          IF (_MessageLevel > E_MessageType.eMessageError)
          THEN
            _stMsg.eType            := E_MessageType.eMessageInfo;
            _stMsg.eSubdevice       := e_Subdevice.Process_ProcessCollector_Cycle;
            _stMsg.iErrorNumber     := _nProcessId;
            _stMsg.sText            := concat(TO_STRING(_stState.State), ': ');
            _stMsg.sText            := concat(_stMsg.sText, TO_STRING(_eStateProgress));
            f_MessageSet(_stMsg);
          END_IF


        E_PROCESS_CTRL.PROCESS_STATIONS_SEND:
          _eCmd                     := _stControl.Cmd;                  // start skipping of process

          LogControl(_eCmd);

          _eStateProgress           := E_PROGRESS.PROGRESS_INIT;        // switch back sub state
          _stState.State            := E_PROCESS_STATE.PROCESS_STATIONS_OUTFEED;

          IF (_MessageLevel > E_MessageType.eMessageError)
          THEN
            _stMsg.eType            := E_MessageType.eMessageInfo;
            _stMsg.eSubdevice       := e_Subdevice.Process_ProcessCollector_Cycle;
            _stMsg.iErrorNumber     := _nProcessId;
            _stMsg.sText            := concat(TO_STRING(_stState.State), ': ');
            _stMsg.sText            := concat(_stMsg.sText, TO_STRING(_eStateProgress));
            f_MessageSet(_stMsg);
          END_IF
      END_CASE
    END_CASE
END_CASE
//-------------------------------------------------------------------------------------------------
//-------------------------------------------------------------------------------------------------
CASE _stState.State
OF
  //-----------------------------------------------------------------------------------------------
  E_PROCESS_STATE.PROCESS_STATIONS_NEST:  // wait state before movers are positioned to next nest
    //-------------------------------------------------------------------------
    CASE _eStateProgress
    OF
      E_PROGRESS.PROGRESS_INIT:
        IF (_wStateNest = _wActivateStation)  // ...to include everyone
        THEN
          _eStateProgress           := E_PROGRESS.PROGRESS_BUSY;

          IF (_MessageLevel > E_MessageType.eMessageWarning)
          THEN
            _stMsg.eType            := E_MessageType.eMessageInfo;
            _stMsg.eSubdevice       := e_Subdevice.Process_ProcessCollector_Cycle;
            _stMsg.iErrorNumber     := _wStateNest;
            _stMsg.sText            := concat('_wStateNest: ', BitsToString(_wStateNest));
            _stMsg.sText            := concat(_stMsg.sText, ': ');
            _stMsg.sText            := concat(_stMsg.sText, TO_STRING(_eStateProgress));
            f_MessageSet(_stMsg);
          END_IF
        END_IF
    END_CASE
    //-------------------------------------------------------------------------
    CASE _eStateProgress
    OF
      E_PROGRESS.PROGRESS_BUSY:
      CASE _stControl.Cmd
      OF
        E_PROCESS_CTRL.PROCESS_STATIONS_ENTER:
          _eCmd                     := _stControl.Cmd;                  // copy command to start movement to next nest

          LogControl(_eCmd);

          _eStateProgress           := E_PROGRESS.PROGRESS_INIT;        // switch back sub state
          _stState.State            := E_PROCESS_STATE.PROCESS_START;

          IF (_MessageLevel > E_MessageType.eMessageWarning)
          THEN
            _stMsg.eType            := E_MessageType.eMessageInfo;
            _stMsg.eSubdevice       := e_Subdevice.Process_ProcessCollector_Cycle;
            _stMsg.iErrorNumber     := _nProcessId;
            _stMsg.sText            := concat(TO_STRING(_stState.State), ': ');
            _stMsg.sText            := concat(_stMsg.sText, TO_STRING(_eStateProgress));
            f_MessageSet(_stMsg);
          END_IF
      END_CASE
    END_CASE
END_CASE
//-------------------------------------------------------------------------------------------------
//-------------------------------------------------------------------------------------------------
CASE _stState.State
OF
  //-----------------------------------------------------------------------------------------------
  E_PROCESS_STATE.PROCESS_START:    // wait state for movers to arrive
    //-------------------------------------------------------------------------
    CASE _eStateProgress
    OF
      E_PROGRESS.PROGRESS_INIT:
        IF (_wStateStart = _wActivateStation)  
          // all active XtsStations have mover in standstill after infeed, 
          // process handshake may now start
        THEN
          // movers have arrived and are in standstill
          _eStateProgress           := E_PROGRESS.PROGRESS_BUSY;

          IF (_MessageLevel > E_MessageType.eMessageInfo)
          THEN
            _stMsg.eType            := E_MessageType.eMessageVerbose;
            _stMsg.eSubdevice       := e_Subdevice.Process_ProcessCollector_Cycle;
            _stMsg.iErrorNumber     := _wStateStart;
            _stMsg.sText            := concat('_wStateStart: ', BitsToString(_wStateStart));
            _stMsg.sText            := concat(_stMsg.sText, ': ');
            _stMsg.sText            := concat(_stMsg.sText, TO_STRING(_eStateProgress));
            f_MessageSet(_stMsg);
          END_IF
        END_IF
    END_CASE
    //-------------------------------------------------------------------------
    CASE _eStateProgress
    OF
      E_PROGRESS.PROGRESS_BUSY:
      CASE _stControl.Cmd
      OF
        E_PROCESS_CTRL.PROCESS_START,
        E_PROCESS_CTRL.PROCESS_DONE,
        E_PROCESS_CTRL.PROCESS_STATIONS_OUTFEED:
          _eCmd                     := E_PROCESS_CTRL.PROCESS_DONE;     // first handshake for starting process

          LogControl(_eCmd);

          _eStateProgress           := E_PROGRESS.PROGRESS_INIT;        // switch back sub state
          _stState.State            := E_PROCESS_STATE.PROCESS_DONE;

          IF (_MessageLevel > E_MessageType.eMessageWarning)
          THEN
            _stMsg.eType            := E_MessageType.eMessageInfo;
            _stMsg.eSubdevice       := e_Subdevice.Process_ProcessCollector_Cycle;
            _stMsg.iErrorNumber     := _nProcessId;
            _stMsg.sText            := concat(TO_STRING(_stState.State), ': ');
            _stMsg.sText            := concat(_stMsg.sText, TO_STRING(_eStateProgress));
            f_MessageSet(_stMsg);
          END_IF
      END_CASE
    END_CASE
END_CASE
//-------------------------------------------------------------------------------------------------
//-------------------------------------------------------------------------------------------------
CASE _stState.State
OF
  E_PROCESS_STATE.PROCESS_DONE:     // wait state for process done
    //-------------------------------------------------------------------------
    CASE _eStateProgress
    OF
      E_PROGRESS.PROGRESS_INIT:
        IF (_wStateDone = _wActivateStation)
        THEN
          // first handshake done
          _eStateProgress           := E_PROGRESS.PROGRESS_BUSY;

          IF (_MessageLevel > E_MessageType.eMessageInfo)
          THEN
            _stMsg.eType            := E_MessageType.eMessageVerbose;
            _stMsg.eSubdevice       := e_Subdevice.Process_ProcessCollector_Cycle;
            _stMsg.iErrorNumber     := _wStateDone;
            _stMsg.sText            := concat('_wStateDone: ', BitsToString(_wStateDone));
            _stMsg.sText            := concat(_stMsg.sText, ': ');
            _stMsg.sText            := concat(_stMsg.sText, TO_STRING(_eStateProgress));
            f_MessageSet(_stMsg);
          END_IF
        END_IF
    END_CASE
    //-------------------------------------------------------------------------
    CASE _eStateProgress
    OF
      E_PROGRESS.PROGRESS_BUSY:
      CASE _stControl.Cmd
      OF
        E_PROCESS_CTRL.PROCESS_DONE,
        E_PROCESS_CTRL.PROCESS_STATIONS_OUTFEED:
          _eCmd                     := _stControl.Cmd;                  // second handshake for finishing process

          LogControl(_eCmd);

          _eStateProgress           := E_PROGRESS.PROGRESS_CHECK;       // check mover after process done
      END_CASE
    //-------------------------------------------------------------------------
      E_PROGRESS.PROGRESS_CHECK:
        IF (_wStateNest > 0)        // mover has to be worked again
        THEN
          _eStateProgress           := E_PROGRESS.PROGRESS_INIT;        // switch back sub state
          _stState.State            := E_PROCESS_STATE.PROCESS_STATIONS_NEST;

          IF (_MessageLevel > E_MessageType.eMessageInfo)
          THEN
            _stMsg.eType            := E_MessageType.eMessageVerbose;
            _stMsg.eSubdevice       := e_Subdevice.Process_ProcessCollector_Cycle;
            _stMsg.iErrorNumber     := _nProcessId;
            _stMsg.sText            := concat(TO_STRING(_stState.State), ': ');
            _stMsg.sText            := concat(_stMsg.sText, TO_STRING(_eStateProgress));
            f_MessageSet(_stMsg);
          END_IF

        ELSIF (_wStateOut > 0)      // mover has to leave
        THEN
          _eStateProgress           := E_PROGRESS.PROGRESS_INIT;        // switch back sub state
          _stState.State            := E_PROCESS_STATE.PROCESS_STATIONS_OUTFEED;

          IF (_MessageLevel > E_MessageType.eMessageInfo)
          THEN
            _stMsg.eType            := E_MessageType.eMessageVerbose;
            _stMsg.eSubdevice       := e_Subdevice.Process_ProcessCollector_Cycle;
            _stMsg.iErrorNumber     := _nProcessId;
            _stMsg.sText            := concat(TO_STRING(_stState.State), ': ');
            _stMsg.sText            := concat(_stMsg.sText, TO_STRING(_eStateProgress));
            f_MessageSet(_stMsg);
          END_IF
        END_IF
    END_CASE
END_CASE
//-------------------------------------------------------------------------------------------------
//-------------------------------------------------------------------------------------------------
CASE _stState.State
OF
  E_PROCESS_STATE.PROCESS_STATIONS_OUTFEED:   // wait state before movers are sent out
    //-------------------------------------------------------------------------
    CASE _eStateProgress
    OF
      E_PROGRESS.PROGRESS_INIT:
        IF (_wStateOut = _wActivateStation)
        THEN
          // all active stations want to send out mover
          // now is the time for you to have decided the TargetStation(s) and TargetMask(s)
          _eStateProgress           := E_PROGRESS.PROGRESS_BUSY;

          IF (_MessageLevel > E_MessageType.eMessageInfo)
          THEN
            _stMsg.eType            := E_MessageType.eMessageVerbose;
            _stMsg.eSubdevice       := e_Subdevice.Process_ProcessCollector_Cycle;
            _stMsg.iErrorNumber     := _wStateOut;
            _stMsg.sText            := concat('_wStateOut: ', BitsToString(_wStateOut));
            _stMsg.sText            := concat(_stMsg.sText, ': ');
            _stMsg.sText            := concat(_stMsg.sText, TO_STRING(_eStateProgress));
            f_MessageSet(_stMsg);
          END_IF
        END_IF
    END_CASE
    //-------------------------------------------------------------------------
    CASE _eStateProgress
    OF
      E_PROGRESS.PROGRESS_BUSY:     // now is the time to get/write target data
      CASE _stControl.Cmd
      OF
        E_PROCESS_CTRL.PROCESS_STATIONS_OUTFEED:  // before you start the outfeed of station, get/write target data on the outside. Use properties: TargetIndex; TargetMask
          _eCmd                     := _stControl.Cmd;

          LogControl(_eCmd);

          _eStateProgress           := E_PROGRESS.PROGRESS_CHECK;       // check movers gone

          IF (_MessageLevel > E_MessageType.eMessageError)
          THEN
            _stMsg.eType            := E_MessageType.eMessageInfo;
            _stMsg.eSubdevice       := e_Subdevice.Process_ProcessCollector_Cycle;
            _stMsg.iErrorNumber     := _nProcessId;
            _stMsg.sText            := concat(TO_STRING(_stState.State), ': ');
            _stMsg.sText            := concat(_stMsg.sText, TO_STRING(_eStateProgress));
            f_MessageSet(_stMsg);
          END_IF
      END_CASE
    END_CASE
    //-------------------------------------------------------------------------
    CASE _eStateProgress
    OF
      E_PROGRESS.PROGRESS_CHECK:
        IF (_wStateOut = 0)         // all stations are empty, go back to start new infeed of movers
        THEN
          _eStateProgress           := E_PROGRESS.PROGRESS_INIT;        // switch back sub state
          _stState.State            := E_PROCESS_STATE.PROCESS_DISABLE; // switch back to disabled state

          IF (_MessageLevel > E_MessageType.eMessageInfo)
          THEN
            _stMsg.eType            := E_MessageType.eMessageVerbose;
            _stMsg.eSubdevice       := e_Subdevice.Process_ProcessCollector_Cycle;
            _stMsg.iErrorNumber     := _wStateOut;
            _stMsg.sText            := concat('_wStateOut: ', BitsToString(_wStateOut));
            _stMsg.sText            := concat(_stMsg.sText, ': ');
            _stMsg.sText            := concat(_stMsg.sText, TO_STRING(_eStateProgress));
            f_MessageSet(_stMsg);
          END_IF
        END_IF
    END_CASE
END_CASE
//-------------------------------------------------------------------------------------------------
// _eStateProgress information to process result
//-------------------------------------------------------------------------------------------------
_stState.Result                     := _eStateProgress;
//-------------------------------------------------------------------------------------------------
//-------------------------------------------------------------------------------------------------
// _eCheck information for plausibility checks
//-------------------------------------------------------------------------------------------------
_stState.Check                      := _eCheck;
//-------------------------------------------------------------------------------------------------
//-------------------------------------------------------------------------------------------------
// _eCmd - command switch
//-------------------------------------------------------------------------------------------------
Controls(_eCmd);                    // cyclic call for setting commands on XtsStations in process range
//-------------------------------------------------------------------------------------------------
//-------------------------------------------------------------------------------------------------
END_METHOD

METHOD PUBLIC Init : E_PROGRESS // clears all XtsSubstations, then disables all
VAR_INPUT
  Execute     : BOOL;
END_VAR
VAR_INST
  _nIndexStation        : UINT;
  _nErrorId             : UDINT;
  _eState               : E_PROGRESS;
END_VAR
//-----------------------------------------------------------------------------
IF NOT Execute 
THEN 
	_eState                       := E_PROGRESS.PROGRESS_INIT; 
END_IF 
//-----------------------------------------------------------------------------
IF NOT Check() 
THEN 
	Init                          := E_PROGRESS.PROGRESS_ERROR; 
	RETURN; 
END_IF
//-----------------------------------------------------------------------------
//-----------------------------------------------------------------------------
CASE _eState
OF
  E_PROGRESS.PROGRESS_INIT:
    IF Execute
    THEN
      _nIndexStation            := _nStationLast;
      _nErrorId                 := 0;
      _eState                   := E_PROGRESS.PROGRESS_BUSY;
      memset(ADR(_wTargetMask), 1, SIZEOF(_wTargetMask));

      _eCmd                     := E_PROCESS_CTRL.PROCESS_INIT;
      _stState.State            := E_PROCESS_STATE.PROCESS_INVALID;
      _eStateProgress           := E_PROGRESS.PROGRESS_INVALID;


      _stMsg.eType              := _MessageLevel;

      IF (_MessageLevel = E_MessageType.eMessageVerbose)
      THEN
        _stMsg.eSubdevice       := e_Subdevice.Process_ProcessCollector_Init;
        _stMsg.iErrorNumber     := _nIndexStation;
        _stMsg.sText            := concat('.Init: ', TO_STRING(_eState));
        f_MessageSet(_stMsg);
      END_IF
    END_IF
END_CASE
//-----------------------------------------------------------------------------
//-----------------------------------------------------------------------------
CASE _eState
OF
  E_PROGRESS.PROGRESS_BUSY:
    _stStationCtrl[_nIndexStation].Cmd     := E_STATION_CTRL.STATION_INIT;
    _eState                     := E_PROGRESS.PROGRESS_PREPARE;

    IF (_MessageLevel = E_MessageType.eMessageVerbose)
    THEN
      _stMsg.eSubdevice         := e_Subdevice.Process_ProcessCollector_Init;
      _stMsg.iErrorNumber       := _nIndexStation;
      _stMsg.sText              := concat(TO_STRING(_stStationCtrl[_nIndexStation].Cmd), ': ');
      _stMsg.sText              := concat(_stMsg.sText, TO_STRING(_eState));
      f_MessageSet(_stMsg);
    END_IF

  E_PROGRESS.PROGRESS_PREPARE:
    IF (_nIndexStation < _nStationFirst+1)
    THEN
      _eCmdOld                  :=
      _eCmd                     := E_PROCESS_CTRL.PROCESS_DISABLE;
      _nIndexStation            := _nStationFirst;
      _eState                   := E_PROGRESS.PROGRESS_STARTUP;
    ELSE
      IF (_stStationState[_nIndexStation].State = E_STATION_STATE.STATION_INIT)
      THEN
        _nIndexStation          := _nIndexStation - 1;
        _eState                 := E_PROGRESS.PROGRESS_BUSY;
      ELSE
        _eState                 := E_PROGRESS.PROGRESS_BUSY;
      END_IF
    END_IF

  E_PROGRESS.PROGRESS_STARTUP:
    _stStationCtrl[_nIndexStation].Cmd     := E_STATION_CTRL.STATION_DISABLE;
    _eState                     := E_PROGRESS.PROGRESS_CHECK;

    IF (_MessageLevel = E_MessageType.eMessageVerbose)
    THEN
      _stMsg.eSubdevice         := e_Subdevice.Process_ProcessCollector_Init;
      _stMsg.iErrorNumber       := _nIndexStation;
      _stMsg.sText              := concat(TO_STRING(_stStationCtrl[_nIndexStation].Cmd), ': ');
      _stMsg.sText              := concat(_stMsg.sText, TO_STRING(_eState));
      f_MessageSet(_stMsg);
    END_IF

  E_PROGRESS.PROGRESS_CHECK:
    IF NOT (_nIndexStation > _nStationLast-1)
    THEN
      IF (_stStationState[_nIndexStation].State = E_STATION_STATE.STATION_DISABLE)
      THEN
        _nIndexStation          := _nIndexStation + 1;
        _eState                 := E_PROGRESS.PROGRESS_STARTUP;
      END_IF
    ELSE
      // give back result
      _eState                   := E_PROGRESS.PROGRESS_DONE;

      // where were I?
      IF (_MessageLevel = E_MessageType.eMessageVerbose)
      THEN
        _stMsg.eSubdevice       := e_Subdevice.Process_ProcessCollector_Init;
        _stMsg.iErrorNumber     := _nProcessId;
        _stMsg.sText            := concat('.Clear: ', TO_STRING(_stState.State));
        f_MessageSet(_stMsg);
      END_IF

      // clear Cycle() state machine
      _stState.State            := E_PROCESS_STATE.PROCESS_DISABLE;
      _eStateProgress           := E_PROGRESS.PROGRESS_INIT;

      IF (_MessageLevel = E_MessageType.eMessageVerbose)
      THEN
        // init done
        _stMsg.eSubdevice       := e_Subdevice.Process_ProcessCollector_Init;
        _stMsg.iErrorNumber     := _nProcessId;
        _stMsg.sText            := concat('.Init: ', TO_STRING(_eState));
        f_MessageSet(_stMsg);
      END_IF
    END_IF
END_CASE
//-----------------------------------------------------------------------------
//-----------------------------------------------------------------------------

Init := _eState;
END_METHOD

METHOD PRIVATE LogControl
VAR_INPUT
  Cmd         : E_PROCESS_CTRL;
END_VAR
IF (Cmd <> _eCmdOld)
THEN
  IF (_MessageLevel > E_MessageType.eMessageWarning)
  THEN
    _stMsg.eType                          := E_MessageType.eMessageInfo;
    _stMsg.eSubdevice                     := e_Subdevice.Process_ProcessCollector_Control;
    _stMsg.iErrorNumber                   := _nProcessId;
    _stMsg.sText                          := 'Cmd: ';
    _stMsg.sText                          := concat(_stMsg.sText, TO_STRING(Cmd));
    f_MessageSet(_stMsg);
  END_IF

  CASE Cmd                                               // check process command
  OF
    E_PROCESS_CTRL.PROCESS_ENABLE:
      IF (_MessageLevel = E_MessageType.eMessageVerbose)
      THEN
        _stMsg.eType                      := E_MessageType.eMessageVerbose;
        _stMsg.eSubdevice                 := e_Subdevice.Process_ProcessCollector_Control;
        _stMsg.iErrorNumber               := _wActivateStation;
        _stMsg.sText                      := concat('_wActivateStation: ', BitsToString(_wActivateStation));
        f_MessageSet(_stMsg);
      END_IF
   END_CASE
  _eCmdOld                                := Cmd;
END_IF
END_METHOD

PROPERTY MessageLevel : e_MessageType
GET
MessageLevel := _MessageLevel;
END_GET
SET
VAR
  _ix : uint;
END_VAR
_MessageLevel := MessageLevel;

IF NOT (_eCheck = E_PROCESS_CHECK.CHECK_DONE)
THEN
  RETURN;
ELSE
  FOR _ix := _nStationFirst TO _nStationLast
  DO
    GVL_MSG_XTS.MessageLevelStations[_ix]   := _MessageLevel;
  END_FOR
END_IF
END_SET
END_PROPERTY

PROPERTY MoverCountTotal : udint
GET
MoverCountTotal := _nMoverCountTotal;
END_GET
END_PROPERTY

PROPERTY MoverPerMinute : udint
GET
MoverPerMinute := _AllStationMoverPerMinute;
END_GET
END_PROPERTY

PROPERTY ProcessCtrl : reference to st_process_ctrl
GET
ProcessCtrl REF= _stControl;
END_GET
SET
_stControl ref= ProcessCtrl;
END_SET
END_PROPERTY

PROPERTY ProcessId : E_INSTANCE
GET
Processid := _nProcessId;
END_GET
SET
_nProcessId := ProcessId;
END_SET
END_PROPERTY

PROPERTY ProcessState : reference to st_process_state
GET
ProcessState REF= _stState;
END_GET
SET
_stState ref= ProcessState;
END_SET
END_PROPERTY

PROPERTY TargetIndex : ARRAY[1..SIZEOF(T_PROCESS)*8] OF USINT
GET
TargetIndex := _nTargetIndex;
END_GET
SET
_nTargetIndex := TargetIndex;
END_SET
END_PROPERTY

PROPERTY TargetMask : ARRAY[1..SIZEOF(T_PROCESS)*8] OF BYTE
GET
TargetMask := _wTargetMask;
END_GET
SET
_wTargetMask := TargetMask;
END_SET
END_PROPERTY

METHOD Template : E_PROGRESS
VAR_INPUT
  Execute     : BOOL;
END_VAR
VAR_INST
  _nErrorId   : UDINT;
  _eState     : E_PROGRESS;
END_VAR
//-----------------------------------------------------------------------------
IF NOT Execute 
THEN 
	_eState                       := E_PROGRESS.PROGRESS_INIT; 
END_IF 
//-----------------------------------------------------------------------------
IF NOT Check() 
THEN 
	Template_1                    := E_PROGRESS.PROGRESS_ERROR; 
	RETURN; 
END_IF
//-----------------------------------------------------------------------------
//-----------------------------------------------------------------------------
CASE _eState
OF
  E_PROGRESS.PROGRESS_INIT:
    IF Execute
    THEN
      _nErrorId                 := 0;

      _eState                   := E_PROGRESS.PROGRESS_BUSY;
    END_IF
END_CASE
//-----------------------------------------------------------------------------
//-----------------------------------------------------------------------------
CASE _eState
OF
  E_PROGRESS.PROGRESS_BUSY:
    _eState                     := E_PROGRESS.PROGRESS_PREPARE;
END_CASE
//-----------------------------------------------------------------------------
//-----------------------------------------------------------------------------
CASE _eState
OF
  E_PROGRESS.PROGRESS_PREPARE:

    IF (.Error)
    THEN
      _eState                   := E_PROGRESS.PROGRESS_ERROR;
      _nErrorId                 := 


    ELSIF (.Done)
    THEN
      _eState                   := E_PROGRESS.;

    END_IF
END_CASE
//-----------------------------------------------------------------------------
//-----------------------------------------------------------------------------

Template_1                      := _eState;
END_METHOD

END_FUNCTION_BLOCK
